(* CODESYS project wago_write_local_file_example_v0.0.1.ecp

Project tree, tasks and I/O mapping:
  PFC200_2ETH_RS : 750-8202 PFC200 2ETH RS, WAGO, order no. 0750-8202, version 5.11.1.16
    application Application
      libraries: ; WagoAppFileDir, * (WAGO); VisuDialogs, * (System); WagoSysString, * (WAGO); WagoAppString, * (WAGO); WagoTypesCommon, * (WAGO)
      task PLC_Task (cyclic, interval t#50ms, priority 15) calls PLC_PRG
      task VISU_TASK (cyclic, interval 100 ms, priority 15) calls VisuElems.Visu_Prg
      program PLC_PRG [ST]
      visualisation Visualization
    DeviceAdapter
    Kbus : Kbus, WAGO, version 1.4.0.2
        unmapped channels: K-BUS diagnostics
    MODBUS
      MODBUS : MODBUS, WAGO, order no. n/a, version 1.1.1.15
    Serial
      COM1 : COM1, WAGO, version 0.0.0.19
  text list GlobalTextList
*)

// PFC200_2ETH_RS/Application/PLC_PRG
PROGRAM PLC_PRG
VAR
	Progress		: INT;
	File			: fbGeneralFile;
	xWriteFile		: BOOL;
	
	sStringFromVisu	: STRING := 'Hello World!';
	sStringToWrite	: STRING;
	xFileOpenBtn	: BOOL;
	xFileWriteBtn	: BOOL;
	xFileCloseBtn	: BOOL;
END_VAR

//create the written line with a newline char
sStringToWrite := CONCAT(sStringFromVisu, ASCIIBYTE_TO_STRING(16#0A));

//open the file (create if doesnt exist)
IF xFileOpenBtn THEN
	File.Open('testfile.csv', FAM_APPEND, 0, FALSE);
	IF File.xTerminated THEN
		xFileOpenBtn := FALSE;
	END_IF
END_IF

//write the string
IF xFileWriteBtn THEN
	File.WriteString(sStringToWrite);
	IF File.xTerminated THEN
		xFileWriteBtn := FALSE;
	END_IF
END_IF

//close the file
IF xFileCloseBtn THEN
	File.Close();
	IF File.xTerminated THEN
		xFileCloseBtn := FALSE;
	END_IF
END_IF

END_PROGRAM

// PFC200_2ETH_RS/Application/Visualization
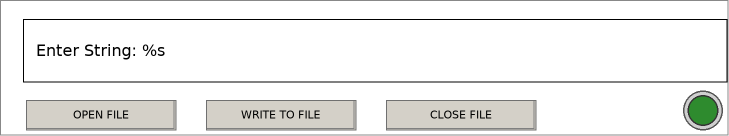
VISUALIZATION Visualization  // 729x136
    Rectangle (23,19 704x63), "Enter String: %s", text variable: PLC_PRG.sStringFromVisu
        OnMouseDown: write the text variable via Default
    Button (26,100 150x30), "OPEN FILE"
        toggle PLC_PRG.xFileOpenBtn
    Button (206,100 150x30), "WRITE TO FILE"
        toggle PLC_PRG.xFileWriteBtn
    Button (386,100 150x30), "CLOSE FILE"
        toggle PLC_PRG.xFileCloseBtn
    Lamp1 (680,87 46x47), variable: PLC_PRG.File.xIsOpen, style: Lamp-Lamp1-Green
END_VISUALIZATION
